// TIA Portal V17 export
// export: Created 2025-06-25T13:13:02.579862Z, ExportSetting WithDefaults, DisplayName Totally Integrated Automation Portal, DisplayVersion V17 Update 8, DisplayName TIA Portal Openness, DisplayVersion V17 Update 8, DisplayName TIA Portal Version Control Interface, DisplayVersion V17, DisplayName STEP 7 Professional, DisplayVersion V17 Update 8, DisplayName STEP 7 Safety, DisplayVersion V17 Update 6, DisplayName WinCC Advanced, DisplayVersion V17 Update 8
ORGANIZATION_BLOCK "Main_Cyclic"   // OB35, FBD, CyclicInterrupt
TITLE = Realtime task
{ S7_Optimized_Access := 'TRUE' }
VERSION : 0.1
// stored: AutoNumber false, IsIECCheckEnabled false, SetENOAutomatically false
   VAR_INPUT
      Initial_Call : Bool;
      Event_Count : Int;
   END_VAR
BEGIN

REGION Network 1
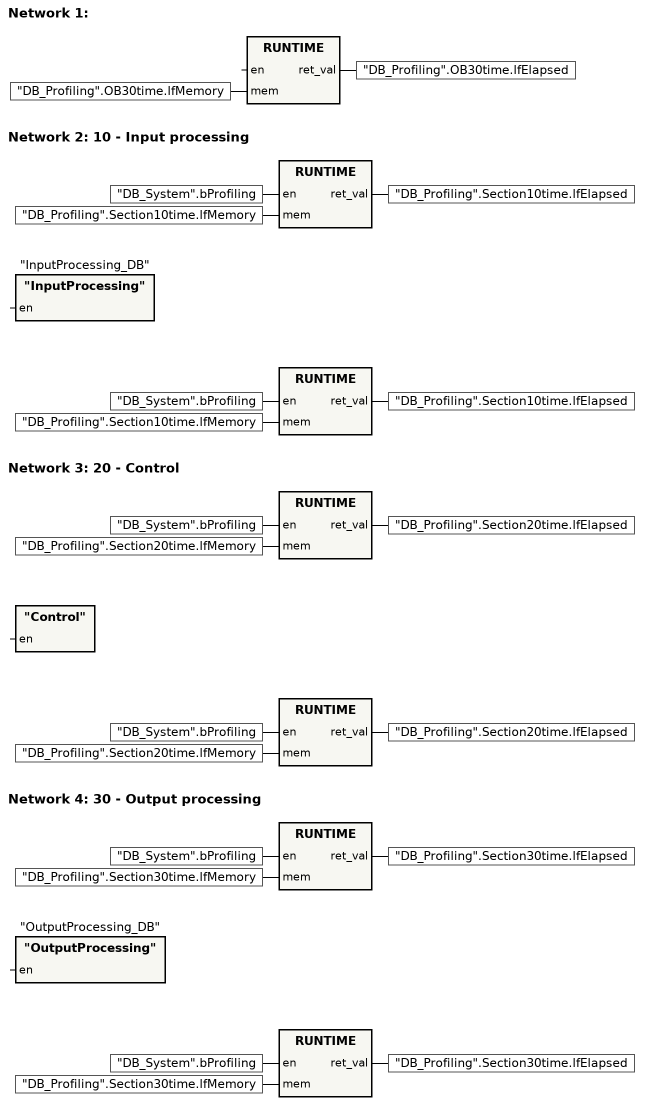
   // no SCL statement known for Runtime: written as a call
   "DB_Profiling".OB30time.lfElapsed := Runtime(mem := "DB_Profiling".OB30time.lfMemory);
END_REGION

REGION Network 2: 10 - Input processing
   // no SCL statement known for Runtime: written as a call
   IF "DB_System".bProfiling THEN
       "DB_Profiling".Section10time.lfElapsed := Runtime(mem := "DB_Profiling".Section10time.lfMemory);
   END_IF;
   "InputProcessing_DB"();   // "InputProcessing"
   IF "DB_System".bProfiling THEN
       "DB_Profiling".Section10time.lfElapsed := Runtime(mem := "DB_Profiling".Section10time.lfMemory);
   END_IF;
END_REGION

REGION Network 3: 20 - Control
   // no SCL statement known for Runtime: written as a call
   IF "DB_System".bProfiling THEN
       "DB_Profiling".Section20time.lfElapsed := Runtime(mem := "DB_Profiling".Section20time.lfMemory);
   END_IF;
   "Control"();
   IF "DB_System".bProfiling THEN
       "DB_Profiling".Section20time.lfElapsed := Runtime(mem := "DB_Profiling".Section20time.lfMemory);
   END_IF;
END_REGION

REGION Network 4: 30 - Output processing
   // no SCL statement known for Runtime: written as a call
   IF "DB_System".bProfiling THEN
       "DB_Profiling".Section30time.lfElapsed := Runtime(mem := "DB_Profiling".Section30time.lfMemory);
   END_IF;
   "OutputProcessing_DB"();   // "OutputProcessing"
   IF "DB_System".bProfiling THEN
       "DB_Profiling".Section30time.lfElapsed := Runtime(mem := "DB_Profiling".Section30time.lfMemory);
   END_IF;
END_REGION

REGION Network 5: 40 - Alarms
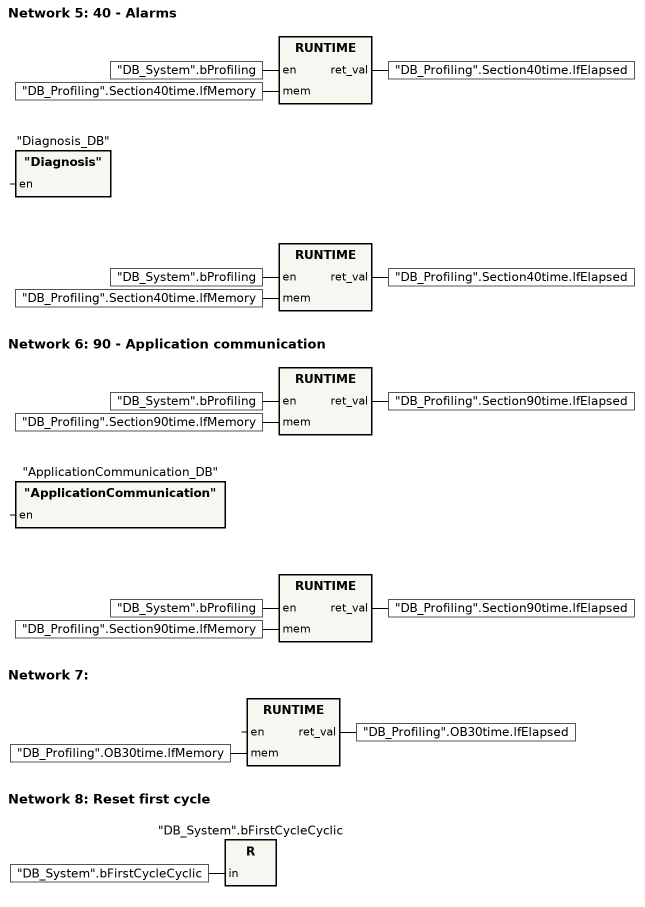
   // no SCL statement known for Runtime: written as a call
   IF "DB_System".bProfiling THEN
       "DB_Profiling".Section40time.lfElapsed := Runtime(mem := "DB_Profiling".Section40time.lfMemory);
   END_IF;
   "Diagnosis_DB"();   // "Diagnosis"
   IF "DB_System".bProfiling THEN
       "DB_Profiling".Section40time.lfElapsed := Runtime(mem := "DB_Profiling".Section40time.lfMemory);
   END_IF;
END_REGION

REGION Network 6: 90 - Application communication
   // Exchange data with the Application PLC
   // no SCL statement known for Runtime: written as a call
   IF "DB_System".bProfiling THEN
       "DB_Profiling".Section90time.lfElapsed := Runtime(mem := "DB_Profiling".Section90time.lfMemory);
   END_IF;
   "ApplicationCommunication_DB"();   // "ApplicationCommunication"
   IF "DB_System".bProfiling THEN
       "DB_Profiling".Section90time.lfElapsed := Runtime(mem := "DB_Profiling".Section90time.lfMemory);
   END_IF;
END_REGION

REGION Network 7
   // no SCL statement known for Runtime: written as a call
   "DB_Profiling".OB30time.lfElapsed := Runtime(mem := "DB_Profiling".OB30time.lfMemory);
END_REGION

REGION Network 8: Reset first cycle
   // This network must be the last one in the program
   IF "DB_System".bFirstCycleCyclic THEN "DB_System".bFirstCycleCyclic := FALSE; END_IF;
END_REGION
END_ORGANIZATION_BLOCK
